// TwinCAT 3 PLC project mobject_promises
// Title: mobject-promises
// Company: mobject
// Author: mobject dev team
// ProjectVersion: 0.1.0
// ProgramVersion: 3.1.4024.0
// libraries:
//   mobject-collections, * (mobject)
//   mobject-disposable, * (mobject)
//   Tc2_System, * (Beckhoff Automation GmbH)
// project tree:
//   Interfaces/ I_Promise.TcIO
//   Promise/ Promise.TcPOU
//   _Internal/Context/ I_PromiseContext.TcIO, PromiseContext.TcPOU

// ---- Interfaces/I_Promise.TcIO
{attribute 'linkalways'} 
INTERFACE I_Promise EXTENDS I_Disposable

PROPERTY PUBLIC Pending : BOOL
GET
END_GET
END_PROPERTY

PROPERTY Rejected : BOOL
GET
END_GET
END_PROPERTY

PROPERTY RejectedReason : T_MAXSTRING
GET
END_GET
END_PROPERTY

PROPERTY Resolved : BOOL
GET
END_GET
END_PROPERTY

METHOD PUBLIC TryGetResult : BOOL
VAR_INPUT
	Destination : ANY;
END_VAR
END_METHOD

METHOD PUBLIC TryGetResultTo : BOOL
VAR_INPUT
	DestinationAddress : PVOID;
	DestinationSize : UDINT;
END_VAR
END_METHOD

END_INTERFACE

// ---- _Internal/Context/I_PromiseContext.TcIO
{attribute 'linkalways'} 
INTERFACE I_PromiseContext

METHOD PUBLIC Reject
VAR_INPUT
	Reason : T_MAXSTRING;
END_VAR
END_METHOD

METHOD PUBLIC Resolve
VAR_INPUT
END_VAR
END_METHOD

METHOD PUBLIC ResolveWith
VAR_INPUT
	Value : ANY;
END_VAR
END_METHOD

METHOD PUBLIC TryGetEntity : BOOL
VAR_INPUT
	Key : T_MAXSTRING;
	Destination	: ANY;
END_VAR
END_METHOD

METHOD PUBLIC TryGetEntityTo : BOOL
VAR_INPUT
	Key : T_MAXSTRING;
	DestinationAddress : PVOID;
	DestinationSize : UDINT;
END_VAR
END_METHOD

METHOD PUBLIC TrySetEntity : BOOL
VAR_INPUT
	Key : T_MAXSTRING;
	Value : ANY;
END_VAR
END_METHOD

END_INTERFACE

// ---- Promise/Promise.TcPOU
{attribute 'linkalways'} 
{attribute 'no_explicit_call' := 'This FB is a CLASS and must be accessed using methods or properties'}
{attribute 'enable_dynamic_creation'}
FUNCTION_BLOCK Promise EXTENDS Disposable IMPLEMENTS I_Promise
VAR
	context : PromiseContext;
END_VAR

PROPERTY PUBLIC Ctx : I_PromiseContext
GET
Ctx := context;
END_GET
END_PROPERTY

PROPERTY PUBLIC Pending : BOOL
GET
Pending := context.Pending;
END_GET
END_PROPERTY

PROPERTY Rejected : BOOL
GET
Rejected := context.Rejected;
END_GET
END_PROPERTY

PROPERTY RejectedReason : T_MAXSTRING
GET
RejectedReason := context.RejectedReason;
END_GET
END_PROPERTY

PROPERTY Resolved : BOOL
GET
Resolved := context.Resolved;
END_GET
END_PROPERTY

METHOD PUBLIC TryGetResult : BOOL
VAR_INPUT
	Destination : ANY;
END_VAR
TryGetResult := context.TryGetResult(Destination);
END_METHOD

METHOD PUBLIC TryGetResultTo : BOOL
VAR_INPUT
	DestinationAddress : PVOID;
	DestinationSize : UDINT;
END_VAR
TryGetResultTo := context.TryGetResultTo(DestinationAddress,DestinationSize);
END_METHOD

END_FUNCTION_BLOCK

// ---- _Internal/Context/PromiseContext.TcPOU
{attribute 'linkalways'} 
{attribute 'no_explicit_call' := 'This FB is a CLASS and must be accessed using methods or properties'}
{attribute 'enable_dynamic_creation'}
FUNCTION_BLOCK PromiseContext IMPLEMENTS I_PromiseContext
VAR
	state : (PROMISE_PENDING, PROMISE_REJECTED, PROMISE_RESOLVED);
	reason : T_MAXSTRING;
	entities : Dictionary;
	pBuffer : POINTER TO BYTE;
	bufferSize : UDINT;
END_VAR

METHOD PRIVATE CopyBufferToDestination
VAR_INPUT
	DestinationAddress : PVOID;
END_VAR
MEMCPY(DestinationAddress, pBuffer, bufferSize);
END_METHOD

METHOD PRIVATE CopySourceToBuffer
VAR_INPUT
	SourceAddress : PVOID;
END_VAR
MEMCPY(pBuffer, SourceAddress, bufferSize);
END_METHOD

METHOD PRIVATE CreateBuffer
VAR_INPUT
	SizeInBytes : UDINT;
END_VAR
bufferSize := SizeInBytes;
pBuffer := __NEW(BYTE, SizeInBytes);
END_METHOD

METHOD PRIVATE DestroyBuffer
VAR_INPUT
END_VAR
IF pBuffer = 0 THEN
	RETURN;
END_IF

__DELETE(pBuffer);
bufferSize := 0;
END_METHOD

METHOD FB_exit : BOOL
VAR_INPUT
	bInCopyCode : BOOL; // if TRUE, the exit method is called for exiting an instance that is copied afterwards (online change).
END_VAR
IF bInCopyCode THEN
	RETURN;
END_IF

DestroyBuffer();
END_METHOD

PROPERTY PUBLIC Pending : BOOL
GET
Pending := state = PROMISE_PENDING;
END_GET
END_PROPERTY

METHOD PUBLIC Reject
VAR_INPUT
	Reason : T_MAXSTRING;
END_VAR
IF NOT Pending THEN
	RETURN;
END_IF

THIS^.reason := Reason;
state := PROMISE_REJECTED;
END_METHOD

PROPERTY Rejected : BOOL
GET
Rejected := state = PROMISE_REJECTED;
END_GET
END_PROPERTY

PROPERTY RejectedReason : T_MAXSTRING
GET
RejectedReason := reason;
END_GET
END_PROPERTY

METHOD PUBLIC Resolve
VAR_INPUT
END_VAR
IF NOT Pending THEN
	RETURN;
END_IF

state := PROMISE_RESOLVED;
END_METHOD

PROPERTY Resolved : BOOL
GET
Resolved := state = PROMISE_RESOLVED;
END_GET
END_PROPERTY

METHOD PUBLIC ResolveWith
VAR_INPUT
	Value : ANY;
END_VAR
IF NOT Pending THEN
	RETURN;
END_IF

state := PROMISE_RESOLVED;
CreateBuffer(DINT_TO_UDINT(Value.diSize));
CopySourceToBuffer(Value.pValue);
END_METHOD

METHOD PUBLIC TryGetEntity : BOOL
VAR_INPUT
	Key : T_MAXSTRING;
	Destination	: ANY;
END_VAR
TryGetEntity := entities.TryGetValue(Key, Destination);
END_METHOD

METHOD PUBLIC TryGetEntityTo : BOOL
VAR_INPUT
	Key : T_MAXSTRING;
	DestinationAddress : PVOID;
	DestinationSize : UDINT;
END_VAR
TryGetEntityTo := entities.TryGetValueTo(Key, DestinationAddress, DestinationSize);
END_METHOD

METHOD PUBLIC TryGetResult : BOOL
VAR_INPUT
	Destination : ANY;
END_VAR
IF NOT Resolved THEN
	RETURN;
END_IF

TryGetResult := TryGetResultTo(Destination.pValue, DINT_TO_UDINT(Destination.diSize));
END_METHOD

METHOD PUBLIC TryGetResultTo : BOOL
VAR_INPUT
	DestinationAddress : PVOID;
	DestinationSize : UDINT;
END_VAR
IF NOT Resolved THEN
	RETURN;
END_IF

IF pBuffer = 0 THEN
	RETURN;
END_IF

IF bufferSize <> DestinationSize THEN
	RETURN;
END_IF

CopyBufferToDestination(DestinationAddress);
TryGetResultTo := TRUE;
END_METHOD

METHOD PUBLIC TrySetEntity : BOOL
VAR_INPUT
	Key : T_MAXSTRING;
	Value : ANY;
END_VAR
TrySetEntity := entities.TryAdd(Key, Value);
END_METHOD

END_FUNCTION_BLOCK
